RoboDK station: robodkiiwa14r820.rdk

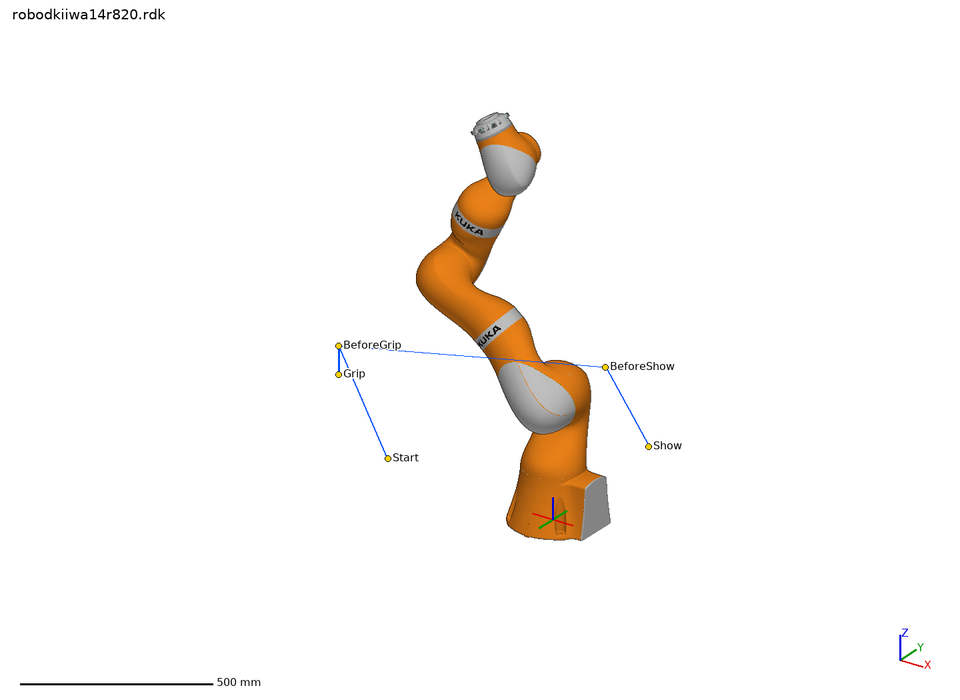
[picture v0: the station drawn from its stored meshes, robots at their saved joint values, targets as dots, program paths as lines]
Station bannerrobodk (saved by RoboDK 5.0.0). Poses are relative to the parent item; angles as X-Y-Z fixed-axis rotations.
Station parameters (name, value as stored): IO_5, 1, Grip, 0
  - frame KUKA LBR iiwa 14 R820 Base at (0, 0, 0) mm, rotated rx 0 ry 0 rz 180 deg
    - robot KUKA LBR iiwa 14 R820: 7 axes, payload 14 kg, reach 1180 mm, repeatability 0.15 mm, weight 29.9 kg
        modified DH rows (alpha deg, a mm, theta deg, d mm): 0, 0, 0, 360; -90, 0, 0, 0; 90, 0, 0, 420; -90, 0, 0, 0; 90, 0, 0, 400; -90, 0, 0, 0; 90, 0, 0, 90
        joint limits [-170, -120, -170, -120, -170, -120, -175] to [170, 120, 170, 120, 170, 120, 175]; home [0, 0, 0, -90, 0, 0, 0]; saved at [3.543, 48.145, 0, -74.39, 0, 57.465, -86.457]
  - program Prog1 (18 instructions, listed below)
  - frame Programm at (0, 0, 0) mm
    - target Grip (Cartesian target) at (-648.81, -40.18, 252.08) mm, rotated rx -180 ry 0 rz 90 deg; joints [3.543, 55.111, 0, -75.083, 0, 49.806, -86.457] of KUKA LBR iiwa 14 R820
    - target BeforeShow (Cartesian target) at (374.91, -298.84, 663.37) mm, rotated rx 51.2 ry 1.22 rz 98.99 deg; joints [134.52, 9.946, 0, -104.683, 139.577, 81.901, -42.43] of KUKA LBR iiwa 14 R820
    - target BeforeGrip (Cartesian target) at (-648.81, -40.18, 335.11) mm, rotated rx 180 ry 0 rz 90 deg; joints [3.543, 48.145, 0, -74.39, 0, 57.465, -86.457] of KUKA LBR iiwa 14 R820
    - target Show (Cartesian target) at (610.53, -440.17, 557.47) mm, rotated rx -149.25 ry 1.8 rz -104.16 deg; joints [-37.339, -47.794, 0, 43.262, 14.89, -61.632, 63.403] of KUKA LBR iiwa 14 R820
    - target Start (Cartesian target) at (-13.03, -726.76, 463.23) mm, rotated rx -161.94 ry 4.4 rz -169.92 deg; joints [88.007, 47.932, 0, -55.491, 9.04, 59.995, -104.756] of KUKA LBR iiwa 14 R820
    - target Target 6 (Cartesian target) at (-13.03, -726.76, 463.23) mm, rotated rx -161.94 ry 4.4 rz -169.92 deg; joints [88.007, 47.932, 0, -55.491, 9.04, 59.995, -104.756] of KUKA LBR iiwa 14 R820
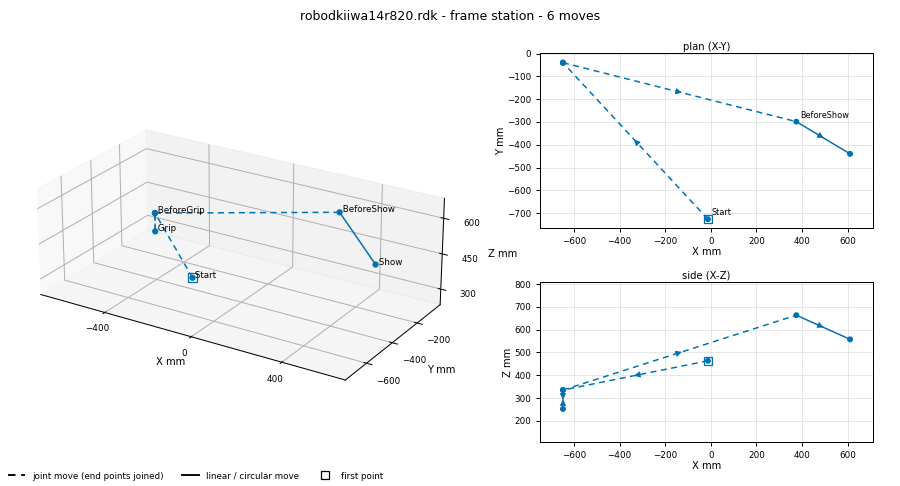
[picture p0: tool path of robodkiiwa14r820.rdk in frame station, 6 of 6 moves have a stored position in this frame; points joined in program order, loops and branches not executed]

--- program Prog1 (robot KUKA LBR iiwa 14 R820) ---
  Set Ref.: Programm
  Set Grip=1
  MoveJ (Start)
  Set IO_5=1
  MoveJ (BeforeGrip)
  Set Grip=0
  Pause 500 ms
  MoveJ (Grip)
  Set Grip=1
  Set IO_5=0
  Pause 500 ms
  MoveJ (BeforeGrip)
  MoveJ (BeforeShow)
  Pause 1.0 s
  MoveL (Show)
  Pause 4.0 s
  Set Grip=0
  Pause 500 ms
